	    ELSE (*Not External Control*)
	        IF Robot.Outputs.MotionControl.MoveID = 32120 THEN
	            Robot.Outputs.MotionControl.MoveID := 32121;
	        ELSIF Robot.Outputs.MotionControl.MoveID = 32121 THEN
	            Robot.Outputs.MotionControl.MoveID := 32120;
	        ELSIF Robot.Outputs.MotionControl.MoveID <> 32120 OR Robot.Outputs.MotionControl.MoveID <> 32121 THEN
	            Robot.Outputs.MotionControl.MoveID := 32120;
	        END_IF;
	        Sent := TRUE;
	    END_IF;
	END_IF;

	(* Check if command has been sent, if so, check if it was received *)
	IF Sent AND
	    Robot.Outputs.MotionCommand.MoveCommand = EnumToNum(Meca500Cmd#SetCartAcc) AND
	    Robot.Outputs.MotionCommand.MoveSubIndex001 = Output_Params[1] AND 
		Robot.Outputs.MotionCommand.MoveSubIndex002 = Output_Params[2] AND 
		Robot.Outputs.MotionCommand.MoveSubIndex003 = Output_Params[3] AND 
		Robot.Outputs.MotionCommand.MoveSubIndex004 = Output_Params[4] AND 
		Robot.Outputs.MotionCommand.MoveSubIndex005 = Output_Params[5] AND 
		Robot.Outputs.MotionCommand.MoveSubIndex006 = Output_Params[6] AND
		Robot.Inputs.Motion.MoveID = Robot.Outputs.MotionControl.MoveID 
	THEN
		 Buffered := TRUE;
	END_IF;


	(*If External _Move ID is equal to Internal, raise an error*)
	IF ExternalMoveID = 32120 OR ExternalMoveID = 32121 THEN
	    Error := TRUE;
	END_IF;

	FirstScan := TRUE;
ELSE
	FirstScan := False;
	Sent := FALSE;
	Buffered := FALSE;
END_IF;
END_FUNCTION_BLOCK

FUNCTION_BLOCK Meca500_SetCartAngVel
VAR
    Output_Params : array[1..6] of real;
    FirstScan : BOOL := False;
END_VAR
VAR_INPUT
    Execute : BOOL;
    Velocity_Limit : REAL;
END_VAR
VAR_OUTPUT
    Sent : BOOL;
    Buffered : BOOL;
    Error : BOOL;
END_VAR
VAR_IN_OUT
    Robot : Meca500;
END_VAR
VAR_INPUT
    ExternalStateControl : BOOL;
    ExternalMoveID : UINT;
END_VAR
IF Execute THEN	
	(*Collect Inputs and store them locally*)
	Output_Params[1]:=Velocity_Limit;
	Output_Params[2]:=0;
	Output_Params[3]:=0;
	Output_Params[4]:=0;
	Output_Params[5]:=0;
	Output_Params[6]:=0;

	(* If Values have change, Reinitialise Outputs*)

	IF FirstScan=0 OR 
		Robot.Outputs.MotionCommand.MoveSubIndex001 <> Output_Params[1] OR 
		Robot.Outputs.MotionCommand.MoveSubIndex002 <> Output_Params[2] OR 
		Robot.Outputs.MotionCommand.MoveSubIndex003 <> Output_Params[3] OR
		Robot.Outputs.MotionCommand.MoveSubIndex004 <> Output_Params[4] OR 
		Robot.Outputs.MotionCommand.MoveSubIndex005 <> Output_Params[5] OR 
		Robot.Outputs.MotionCommand.MoveSubIndex006 <> Output_Params[6] 
	THEN
		Buffered := FALSE;
		Sent := FALSE;
	END_IF;


	(*if not in legacy mode, Act Setpoint*)
	IF Robot.Outputs.MotionControl.MoveID <> 0 THEN
	    Robot.Outputs.MotionControl.SetPoint := TRUE;
	END_IF;

	(* To send _Move, send _Move ID *)
	IF NOT Buffered AND NOT Sent THEN
	    
	    Robot.Outputs.MotionCommand.MoveCommand	:= EnumToNum(Meca500Cmd#SetCartAngVel);
	    Robot.Outputs.MotionCommand.MoveSubIndex001 := Output_Params[1];
		Robot.Outputs.MotionCommand.MoveSubIndex002 := Output_Params[2];
		Robot.Outputs.MotionCommand.MoveSubIndex003 := Output_Params[3];
		Robot.Outputs.MotionCommand.MoveSubIndex004 := Output_Params[4];
		Robot.Outputs.MotionCommand.MoveSubIndex005 := Output_Params[5];
		Robot.Outputs.MotionCommand.MoveSubIndex006 := Output_Params[6];
	    
	    IF ExternalStateControl THEN
	        IF ExternalMoveID <> 0 AND ExternalMoveID <> 32100 AND ExternalMoveID <> 32101 THEN
	            Robot.Outputs.MotionControl.MoveID := ExternalMoveID;
	            Sent := TRUE;
	        END_IF;
	        
	    ELSE (*Not External Control*)
	        IF Robot.Outputs.MotionControl.MoveID = 32100 THEN
	            Robot.Outputs.MotionControl.MoveID := 32101;
	        ELSIF Robot.Outputs.MotionControl.MoveID = 32101 THEN
	            Robot.Outputs.MotionControl.MoveID := 32100;
	        ELSIF Robot.Outputs.MotionControl.MoveID <> 32100 OR Robot.Outputs.MotionControl.MoveID <> 32101 THEN
	            Robot.Outputs.MotionControl.MoveID := 32100;
	        END_IF;
	        Sent := TRUE;
	    END_IF;
	END_IF;

	(* Check if command has been sent, if so, check if it was received *)
	IF Sent AND
	    Robot.Outputs.MotionCommand.MoveCommand = EnumToNum(Meca500Cmd#SetCartAngVel) AND
	    Robot.Outputs.MotionCommand.MoveSubIndex001 = Output_Params[1] AND 
		Robot.Outputs.MotionCommand.MoveSubIndex002 = Output_Params[2] AND 
		Robot.Outputs.MotionCommand.MoveSubIndex003 = Output_Params[3] AND 
		Robot.Outputs.MotionCommand.MoveSubIndex004 = Output_Params[4] AND 
		Robot.Outputs.MotionCommand.MoveSubIndex005 = Output_Params[5] AND 
		Robot.Outputs.MotionCommand.MoveSubIndex006 = Output_Params[6] AND
		Robot.Inputs.Motion.MoveID = Robot.Outputs.MotionControl.MoveID 
	THEN
		 Buffered := TRUE;
	END_IF;


	(*If External _Move ID is equal to Internal, raise an error*)
	IF ExternalMoveID = 32100 OR ExternalMoveID = 32101 THEN
	    Error := TRUE;
	END_IF;

	FirstScan := TRUE;
ELSE
	FirstScan := False;
	Sent := FALSE;
	Buffered := FALSE;
END_IF;
END_FUNCTION_BLOCK

FUNCTION_BLOCK Meca500_SetCartLinVel
VAR
    Output_Params : array[1..6] of real;
    FirstScan : BOOL := False;
END_VAR
VAR_INPUT
    Execute : BOOL;
    Velocity_Limit : REAL;
END_VAR
VAR_OUTPUT
    Sent : BOOL;
    Buffered : BOOL;
    Error : BOOL;
END_VAR
VAR_IN_OUT
    Robot : Meca500;
END_VAR
VAR_INPUT
    ExternalStateControl : BOOL;
    ExternalMoveID : UINT;
END_VAR
IF Execute THEN	
	(*Collect Inputs and store them locally*)
	Output_Params[1]:=Velocity_Limit;
	Output_Params[2]:=0;
	Output_Params[3]:=0;
	Output_Params[4]:=0;
	Output_Params[5]:=0;
	Output_Params[6]:=0;

	(* If Values have change, Reinitialise Outputs*)

	IF FirstScan=0 OR 
		Robot.Outputs.MotionCommand.MoveSubIndex001 <> Output_Params[1] OR 
		Robot.Outputs.MotionCommand.MoveSubIndex002 <> Output_Params[2] OR 
		Robot.Outputs.MotionCommand.MoveSubIndex003 <> Output_Params[3] OR
		Robot.Outputs.MotionCommand.MoveSubIndex004 <> Output_Params[4] OR 
		Robot.Outputs.MotionCommand.MoveSubIndex005 <> Output_Params[5] OR 
		Robot.Outputs.MotionCommand.MoveSubIndex006 <> Output_Params[6] 
	THEN
		Buffered := FALSE;
		Sent := FALSE;
	END_IF;


	(*if not in legacy mode, Act Setpoint*)
	IF Robot.Outputs.MotionControl.MoveID <> 0 THEN
	    Robot.Outputs.MotionControl.SetPoint := TRUE;
	END_IF;

	(* To send _Move, send _Move ID *)
	IF NOT Buffered AND NOT Sent THEN
	    
	    Robot.Outputs.MotionCommand.MoveCommand	:= EnumToNum(Meca500Cmd#SetCartLinVel);
	    Robot.Outputs.MotionCommand.MoveSubIndex001 := Output_Params[1];
		Robot.Outputs.MotionCommand.MoveSubIndex002 := Output_Params[2];
		Robot.Outputs.MotionCommand.MoveSubIndex003 := Output_Params[3];
		Robot.Outputs.MotionCommand.MoveSubIndex004 := Output_Params[4];
		Robot.Outputs.MotionCommand.MoveSubIndex005 := Output_Params[5];
		Robot.Outputs.MotionCommand.MoveSubIndex006 := Output_Params[6];
	    
	    IF ExternalStateControl THEN
	        IF ExternalMoveID <> 0 AND ExternalMoveID <> 32110 AND ExternalMoveID <> 32111 THEN
	            Robot.Outputs.MotionControl.MoveID := ExternalMoveID;
	            Sent := TRUE;
	        END_IF;
	        
	    ELSE (*Not External Control*)
	        IF Robot.Outputs.MotionControl.MoveID = 32110 THEN
	            Robot.Outputs.MotionControl.MoveID := 32111;
	        ELSIF Robot.Outputs.MotionControl.MoveID = 32111 THEN
	            Robot.Outputs.MotionControl.MoveID := 32110;
	        ELSIF Robot.Outputs.MotionControl.MoveID <> 32110 OR Robot.Outputs.MotionControl.MoveID <> 32111 THEN
	            Robot.Outputs.MotionControl.MoveID := 32110;
	        END_IF;
	        Sent := TRUE;
	    END_IF;
	END_IF;

	(* Check if command has been sent, if so, check if it was received *)
	IF Sent AND
	    Robot.Outputs.MotionCommand.MoveCommand = EnumToNum(Meca500Cmd#SetCartLinVel) AND
	    Robot.Outputs.MotionCommand.MoveSubIndex001 = Output_Params[1] AND 
		Robot.Outputs.MotionCommand.MoveSubIndex002 = Output_Params[2] AND 
		Robot.Outputs.MotionCommand.MoveSubIndex003 = Output_Params[3] AND 
		Robot.Outputs.MotionCommand.MoveSubIndex004 = Output_Params[4] AND 
		Robot.Outputs.MotionCommand.MoveSubIndex005 = Output_Params[5] AND 
		Robot.Outputs.MotionCommand.MoveSubIndex006 = Output_Params[6] AND
		Robot.Inputs.Motion.MoveID = Robot.Outputs.MotionControl.MoveID 
	THEN
		 Buffered := TRUE;
	END_IF;


	(*If External _Move ID is equal to Internal, raise an error*)
	IF ExternalMoveID = 32110 OR ExternalMoveID = 32111 THEN
	    Error := TRUE;
	END_IF;

	FirstScan := TRUE;
ELSE
	FirstScan := False;
	Sent := FALSE;
	Buffered := FALSE;
END_IF;
END_FUNCTION_BLOCK

FUNCTION_BLOCK Meca500_SetCheckpoint
VAR
    Output_Params : array[1..6] of real;
    FirstScan : BOOL := False;
END_VAR
VAR_INPUT
    Execute : BOOL;
    CheckpointID : REAL;
END_VAR
VAR_OUTPUT
    Sent : BOOL;
    Buffered : BOOL;
    Error : BOOL;
END_VAR
VAR_IN_OUT
    Robot : Meca500;
END_VAR
VAR_INPUT
    ExternalStateControl : BOOL;
    ExternalMoveID : UINT;
END_VAR
IF Execute THEN	
	(*Collect Inputs and store them locally*)
	Output_Params[1]:=CheckpointID;
	Output_Params[2]:=0;
	Output_Params[3]:=0;
	Output_Params[4]:=0;
	Output_Params[5]:=0;
	Output_Params[6]:=0;

	(* If Values have change, Reinitialise Outputs*)

	IF FirstScan=0 OR 
		Robot.Outputs.MotionCommand.MoveSubIndex001 <> Output_Params[1] OR 
		Robot.Outputs.MotionCommand.MoveSubIndex002 <> Output_Params[2] OR 
		Robot.Outputs.MotionCommand.MoveSubIndex003 <> Output_Params[3] OR
		Robot.Outputs.MotionCommand.MoveSubIndex004 <> Output_Params[4] OR 
		Robot.Outputs.MotionCommand.MoveSubIndex005 <> Output_Params[5] OR 
		Robot.Outputs.MotionCommand.MoveSubIndex006 <> Output_Params[6] 
	THEN
		Buffered := FALSE;
		Sent := FALSE;
	END_IF;


	(*if not in legacy mode, Act Setpoint*)
	IF Robot.Outputs.MotionControl.MoveID <> 0 THEN
	    Robot.Outputs.MotionControl.SetPoint := TRUE;
	END_IF;

	(* To send _Move, send _Move ID *)
	IF NOT Buffered AND NOT Sent THEN
	    
	    Robot.Outputs.MotionCommand.MoveCommand	:= EnumToNum(Meca500Cmd#SetCheckpoint);
	    Robot.Outputs.MotionCommand.MoveSubIndex001 := Output_Params[1];
		Robot.Outputs.MotionCommand.MoveSubIndex002 := Output_Params[2];
		Robot.Outputs.MotionCommand.MoveSubIndex003 := Output_Params[3];
		Robot.Outputs.MotionCommand.MoveSubIndex004 := Output_Params[4];
		Robot.Outputs.MotionCommand.MoveSubIndex005 := Output_Params[5];
		Robot.Outputs.MotionCommand.MoveSubIndex006 := Output_Params[6];
	    
	    IF ExternalStateControl THEN
	        IF ExternalMoveID <> 0 AND ExternalMoveID <> 32170 AND ExternalMoveID <> 32171 THEN
	            Robot.Outputs.MotionControl.MoveID := ExternalMoveID;
	            Sent := TRUE;
	        END_IF;
	        
	    ELSE (*Not External Control*)
	        IF Robot.Outputs.MotionControl.MoveID = 32170 THEN
	            Robot.Outputs.MotionControl.MoveID := 32171;
	        ELSIF Robot.Outputs.MotionControl.MoveID = 32171 THEN
	            Robot.Outputs.MotionControl.MoveID := 32170;
	        ELSIF Robot.Outputs.MotionControl.MoveID <> 32170 OR Robot.Outputs.MotionControl.MoveID <> 32171 THEN
	            Robot.Outputs.MotionControl.MoveID := 32170;
	        END_IF;
	        Sent := TRUE;
	    END_IF;
	END_IF;

	(* Check if command has been sent, if so, check if it was received *)
	IF Sent AND
	    Robot.Outputs.MotionCommand.MoveCommand = EnumToNum(Meca500Cmd#SetCheckpoint) AND
	    Robot.Outputs.MotionCommand.MoveSubIndex001 = Output_Params[1] AND 
		Robot.Outputs.MotionCommand.MoveSubIndex002 = Output_Params[2] AND 
		Robot.Outputs.MotionCommand.MoveSubIndex003 = Output_Params[3] AND 
		Robot.Outputs.MotionCommand.MoveSubIndex004 = Output_Params[4] AND 
		Robot.Outputs.MotionCommand.MoveSubIndex005 = Output_Params[5] AND 
		Robot.Outputs.MotionCommand.MoveSubIndex006 = Output_Params[6] AND
		Robot.Inputs.Motion.MoveID = Robot.Outputs.MotionControl.MoveID 
	THEN
		 Buffered := TRUE;
	END_IF;


	(*If External _Move ID is equal to Internal, raise an error*)
	IF ExternalMoveID = 32170 OR ExternalMoveID = 32171 THEN
	    Error := TRUE;
	END_IF;

	FirstScan := TRUE;
ELSE
	FirstScan := False;
	Sent := FALSE;
	Buffered := FALSE;
END_IF;
END_FUNCTION_BLOCK

FUNCTION_BLOCK Meca500_SetConf
VAR
    Output_Params : array[1..6] of real;
    FirstScan : BOOL := False;
END_VAR
VAR_INPUT
    Execute : BOOL;
    Shoulder : REAL;
    Elbow : REAL;
    Wrist : REAL;
END_VAR
VAR_OUTPUT
    Sent : BOOL;
    Buffered : BOOL;
    Error : BOOL;
END_VAR
VAR_IN_OUT
    Robot : Meca500;
END_VAR
VAR_INPUT
    ExternalStateControl : BOOL;
    ExternalMoveID : UINT;
END_VAR
IF Execute THEN	
	(*Collect Inputs and store them locally*)
	Output_Params[1]:=Shoulder;
	Output_Params[2]:=Elbow;
	Output_Params[3]:=Wrist;
	Output_Params[4]:=0;
	Output_Params[5]:=0;
	Output_Params[6]:=0;

	(* If Values have change, Reinitialise Outputs*)

	IF FirstScan=0 OR 
		Robot.Outputs.MotionCommand.MoveSubIndex001 <> Output_Params[1] OR 
		Robot.Outputs.MotionCommand.MoveSubIndex002 <> Output_Params[2] OR 
		Robot.Outputs.MotionCommand.MoveSubIndex003 <> Output_Params[3] OR
		Robot.Outputs.MotionCommand.MoveSubIndex004 <> Output_Params[4] OR 
		Robot.Outputs.MotionCommand.MoveSubIndex005 <> Output_Params[5] OR 
		Robot.Outputs.MotionCommand.MoveSubIndex006 <> Output_Params[6] 
	THEN
		Buffered := FALSE;
		Sent := FALSE;
	END_IF;


	(*if not in legacy mode, Act Setpoint*)
	IF Robot.Outputs.MotionControl.MoveID <> 0 THEN
	    Robot.Outputs.MotionControl.SetPoint := TRUE;
	END_IF;

	(* To send _Move, send _Move ID *)
	IF NOT Buffered AND NOT Sent THEN
	    
	    Robot.Outputs.MotionCommand.MoveCommand	:= EnumToNum(Meca500Cmd#SetConf);
	    Robot.Outputs.MotionCommand.MoveSubIndex001 := Output_Params[1];
		Robot.Outputs.MotionCommand.MoveSubIndex002 := Output_Params[2];
		Robot.Outputs.MotionCommand.MoveSubIndex003 := Output_Params[3];
		Robot.Outputs.MotionCommand.MoveSubIndex004 := Output_Params[4];
		Robot.Outputs.MotionCommand.MoveSubIndex005 := Output_Params[5];
		Robot.Outputs.MotionCommand.MoveSubIndex006 := Output_Params[6];
	    
	    IF ExternalStateControl THEN
	        IF ExternalMoveID <> 0 AND ExternalMoveID <> 32150 AND ExternalMoveID <> 32151 THEN
	            Robot.Outputs.MotionControl.MoveID := ExternalMoveID;
	            Sent := TRUE;
	        END_IF;
	        
	    ELSE (*Not External Control*)
	        IF Robot.Outputs.MotionControl.MoveID = 32150 THEN
	            Robot.Outputs.MotionControl.MoveID := 32151;
	        ELSIF Robot.Outputs.MotionControl.MoveID = 32151 THEN
	            Robot.Outputs.MotionControl.MoveID := 32150;
	        ELSIF Robot.Outputs.MotionControl.MoveID <> 32150 OR Robot.Outputs.MotionControl.MoveID <> 32151 THEN
	            Robot.Outputs.MotionControl.MoveID := 32150;
	        END_IF;
	        Sent := TRUE;
	    END_IF;
	END_IF;

	(* Check if command has been sent, if so, check if it was received *)
	IF Sent AND
	    Robot.Outputs.MotionCommand.MoveCommand = EnumToNum(Meca500Cmd#SetConf) AND
	    Robot.Outputs.MotionCommand.MoveSubIndex001 = Output_Params[1] AND 
		Robot.Outputs.MotionCommand.MoveSubIndex002 = Output_Params[2] AND 
		Robot.Outputs.MotionCommand.MoveSubIndex003 = Output_Params[3] AND 
		Robot.Outputs.MotionCommand.MoveSubIndex004 = Output_Params[4] AND 
		Robot.Outputs.MotionCommand.MoveSubIndex005 = Output_Params[5] AND 
		Robot.Outputs.MotionCommand.MoveSubIndex006 = Output_Params[6] AND
		Robot.Inputs.Motion.MoveID = Robot.Outputs.MotionControl.MoveID 
	THEN
		 Buffered := TRUE;
	END_IF;


	(*If External _Move ID is equal to Internal, raise an error*)
	IF ExternalMoveID = 32150 OR ExternalMoveID = 32151 THEN
	    Error := TRUE;
	END_IF;

	FirstScan := TRUE;
ELSE
	FirstScan := False;
	Sent := FALSE;
	Buffered := FALSE;
END_IF;
END_FUNCTION_BLOCK

FUNCTION_BLOCK Meca500_SetConfTurn
VAR
    Output_Params : array[1..6] of real;
    FirstScan : BOOL := False;
END_VAR
VAR_INPUT
    Execute : BOOL;
    Config : REAL;
END_VAR
VAR_OUTPUT
    Sent : BOOL;
    Buffered : BOOL;
    Error : BOOL;
END_VAR
VAR_IN_OUT
    Robot : Meca500;
END_VAR
VAR_INPUT
    ExternalStateControl : BOOL;
    ExternalMoveID : UINT;
END_VAR
IF Execute THEN	
	(*Collect Inputs and store them locally*)
	Output_Params[1]:=Config;
	Output_Params[2]:=0;
	Output_Params[3]:=0;
	Output_Params[4]:=0;
	Output_Params[5]:=0;
	Output_Params[6]:=0;

	(* If Values have change, Reinitialise Outputs*)

	IF FirstScan=0 OR 
		Robot.Outputs.MotionCommand.MoveSubIndex001 <> Output_Params[1] OR 
		Robot.Outputs.MotionCommand.MoveSubIndex002 <> Output_Params[2] OR 
		Robot.Outputs.MotionCommand.MoveSubIndex003 <> Output_Params[3] OR
		Robot.Outputs.MotionCommand.MoveSubIndex004 <> Output_Params[4] OR 
		Robot.Outputs.MotionCommand.MoveSubIndex005 <> Output_Params[5] OR 
		Robot.Outputs.MotionCommand.MoveSubIndex006 <> Output_Params[6] 
	THEN
		Buffered := FALSE;
		Sent := FALSE;
	END_IF;


	(*if not in legacy mode, Act Setpoint*)
	IF Robot.Outputs.MotionControl.MoveID <> 0 THEN
	    Robot.Outputs.MotionControl.SetPoint := TRUE;
	END_IF;

	(* To send _Move, send _Move ID *)
	IF NOT Buffered AND NOT Sent THEN
	    
	    Robot.Outputs.MotionCommand.MoveCommand	:= EnumToNum(Meca500Cmd#SetConfTurn);
	    Robot.Outputs.MotionCommand.MoveSubIndex001 := Output_Params[1];
		Robot.Outputs.MotionCommand.MoveSubIndex002 := Output_Params[2];
		Robot.Outputs.MotionCommand.MoveSubIndex003 := Output_Params[3];
		Robot.Outputs.MotionCommand.MoveSubIndex004 := Output_Params[4];
		Robot.Outputs.MotionCommand.MoveSubIndex005 := Output_Params[5];
		Robot.Outputs.MotionCommand.MoveSubIndex006 := Output_Params[6];
	    
	    IF ExternalStateControl THEN
	        IF ExternalMoveID <> 0 AND ExternalMoveID <> 32250 AND ExternalMoveID <> 32251 THEN
	            Robot.Outputs.MotionControl.MoveID := ExternalMoveID;
	            Sent := TRUE;
	        END_IF;
	        
	    ELSE (*Not External Control*)
	        IF Robot.Outputs.MotionControl.MoveID = 32250 THEN
	            Robot.Outputs.MotionControl.MoveID := 32251;
	        ELSIF Robot.Outputs.MotionControl.MoveID = 32251 THEN
	            Robot.Outputs.MotionControl.MoveID := 32250;
	        ELSIF Robot.Outputs.MotionControl.MoveID <> 32250 OR Robot.Outputs.MotionControl.MoveID <> 32251 THEN
	            Robot.Outputs.MotionControl.MoveID := 32250;
	        END_IF;
	        Sent := TRUE;
	    END_IF;
	END_IF;

	(* Check if command has been sent, if so, check if it was received *)
	IF Sent AND
	    Robot.Outputs.MotionCommand.MoveCommand = EnumToNum(Meca500Cmd#SetConfTurn) AND
	    Robot.Outputs.MotionCommand.MoveSubIndex001 = Output_Params[1] AND 
		Robot.Outputs.MotionCommand.MoveSubIndex002 = Output_Params[2] AND 
		Robot.Outputs.MotionCommand.MoveSubIndex003 = Output_Params[3] AND 
		Robot.Outputs.MotionCommand.MoveSubIndex004 = Output_Params[4] AND 
		Robot.Outputs.MotionCommand.MoveSubIndex005 = Output_Params[5] AND 
		Robot.Outputs.MotionCommand.MoveSubIndex006 = Output_Params[6] AND
		Robot.Inputs.Motion.MoveID = Robot.Outputs.MotionControl.MoveID 
	THEN
		 Buffered := TRUE;
	END_IF;


	(*If External _Move ID is equal to Internal, raise an error*)
	IF ExternalMoveID = 32250 OR ExternalMoveID = 32251 THEN
	    Error := TRUE;
	END_IF;

	FirstScan := TRUE;
ELSE
	FirstScan := False;
	Sent := FALSE;
	Buffered := FALSE;
END_IF;
END_FUNCTION_BLOCK

FUNCTION_BLOCK Meca500_SetGripperForce
VAR
    Output_Params : array[1..6] of real;
    FirstScan : BOOL := False;
END_VAR
VAR_INPUT
    Execute : BOOL;
    Force : REAL;
END_VAR
VAR_OUTPUT
    Sent : BOOL;
    Buffered : BOOL;
    Error : BOOL;
END_VAR
VAR_IN_OUT
    Robot : Meca500;
END_VAR
VAR_INPUT
    ExternalStateControl : BOOL;
    ExternalMoveID : UINT;
END_VAR
IF Execute THEN	
	(*Collect Inputs and store them locally*)
	Output_Params[1]:=Force;
	Output_Params[2]:=0;
	Output_Params[3]:=0;
	Output_Params[4]:=0;
	Output_Params[5]:=0;
	Output_Params[6]:=0;

	(* If Values have change, Reinitialise Outputs*)

	IF FirstScan=0 OR 
		Robot.Outputs.MotionCommand.MoveSubIndex001 <> Output_Params[1] OR 
		Robot.Outputs.MotionCommand.MoveSubIndex002 <> Output_Params[2] OR 
		Robot.Outputs.MotionCommand.MoveSubIndex003 <> Output_Params[3] OR
		Robot.Outputs.MotionCommand.MoveSubIndex004 <> Output_Params[4] OR 
		Robot.Outputs.MotionCommand.MoveSubIndex005 <> Output_Params[5] OR 
		Robot.Outputs.MotionCommand.MoveSubIndex006 <> Output_Params[6] 
	THEN
		Buffered := FALSE;
		Sent := FALSE;
	END_IF;


	(*if not in legacy mode, Act Setpoint*)
	IF Robot.Outputs.MotionControl.MoveID <> 0 THEN
	    Robot.Outputs.MotionControl.SetPoint := TRUE;
	END_IF;

	(* To send _Move, send _Move ID *)
	IF NOT Buffered AND NOT Sent THEN
	    
	    Robot.Outputs.MotionCommand.MoveCommand	:= EnumToNum(Meca500Cmd#SetGripperForce);
	    Robot.Outputs.MotionCommand.MoveSubIndex001 := Output_Params[1];
		Robot.Outputs.MotionCommand.MoveSubIndex002 := Output_Params[2];
		Robot.Outputs.MotionCommand.MoveSubIndex003 := Output_Params[3];
		Robot.Outputs.MotionCommand.MoveSubIndex004 := Output_Params[4];
		Robot.Outputs.MotionCommand.MoveSubIndex005 := Output_Params[5];
		Robot.Outputs.MotionCommand.MoveSubIndex006 := Output_Params[6];
	    
	    IF ExternalStateControl THEN
	        IF ExternalMoveID <> 0 AND ExternalMoveID <> 32200 AND ExternalMoveID <> 32201 THEN
	            Robot.Outputs.MotionControl.MoveID := ExternalMoveID;
	            Sent := TRUE;
	        END_IF;
	        
	    ELSE (*Not External Control*)
	        IF Robot.Outputs.MotionControl.MoveID = 32200 THEN
	            Robot.Outputs.MotionControl.MoveID := 32201;
	        ELSIF Robot.Outputs.MotionControl.MoveID = 32201 THEN
	            Robot.Outputs.MotionControl.MoveID := 32200;
	        ELSIF Robot.Outputs.MotionControl.MoveID <> 32200 OR Robot.Outputs.MotionControl.MoveID <> 32201 THEN
	            Robot.Outputs.MotionControl.MoveID := 32200;
	        END_IF;
	        Sent := TRUE;
	    END_IF;
	END_IF;

	(* Check if command has been sent, if so, check if it was received *)
	IF Sent AND
	    Robot.Outputs.MotionCommand.MoveCommand = EnumToNum(Meca500Cmd#SetGripperForce) AND
	    Robot.Outputs.MotionCommand.MoveSubIndex001 = Output_Params[1] AND 
		Robot.Outputs.MotionCommand.MoveSubIndex002 = Output_Params[2] AND 
		Robot.Outputs.MotionCommand.MoveSubIndex003 = Output_Params[3] AND 
		Robot.Outputs.MotionCommand.MoveSubIndex004 = Output_Params[4] AND 
		Robot.Outputs.MotionCommand.MoveSubIndex005 = Output_Params[5] AND 
		Robot.Outputs.MotionCommand.MoveSubIndex006 = Output_Params[6] AND
		Robot.Inputs.Motion.MoveID = Robot.Outputs.MotionControl.MoveID 
	THEN
		 Buffered := TRUE;
	END_IF;


	(*If External _Move ID is equal to Internal, raise an error*)
	IF ExternalMoveID = 32200 OR ExternalMoveID = 32201 THEN
	    Error := TRUE;
	END_IF;

	FirstScan := TRUE;
ELSE
	FirstScan := False;
	Sent := FALSE;
	Buffered := FALSE;
END_IF;
END_FUNCTION_BLOCK

FUNCTION_BLOCK Meca500_SetGripperRange
VAR
    Output_Params : array[1..6] of real;
    FirstScan : BOOL := False;
END_VAR
VAR_INPUT
    Execute : BOOL;
    Minimum : REAL;
    Maximum : REAL;
END_VAR
VAR_OUTPUT
    Sent : BOOL;
    Buffered : BOOL;
    Error : BOOL;
END_VAR
VAR_IN_OUT
    Robot : Meca500;
END_VAR
VAR_INPUT
    ExternalStateControl : BOOL;
    ExternalMoveID : UINT;
END_VAR
IF Execute THEN	
	(*Collect Inputs and store them locally*)
	Output_Params[1]:=Minimum;
	Output_Params[2]:=Maximum;
	Output_Params[3]:=0;
	Output_Params[4]:=0;
	Output_Params[5]:=0;
	Output_Params[6]:=0;

	(* If Values have change, Reinitialise Outputs*)

	IF FirstScan=0 OR 
		Robot.Outputs.MotionCommand.MoveSubIndex001 <> Output_Params[1] OR 
		Robot.Outputs.MotionCommand.MoveSubIndex002 <> Output_Params[2] OR 
		Robot.Outputs.MotionCommand.MoveSubIndex003 <> Output_Params[3] OR
		Robot.Outputs.MotionCommand.MoveSubIndex004 <> Output_Params[4] OR 
		Robot.Outputs.MotionCommand.MoveSubIndex005 <> Output_Params[5] OR 
		Robot.Outputs.MotionCommand.MoveSubIndex006 <> Output_Params[6] 
	THEN
		Buffered := FALSE;
		Sent := FALSE;
	END_IF;


	(*if not in legacy mode, Act Setpoint*)
	IF Robot.Outputs.MotionControl.MoveID <> 0 THEN
	    Robot.Outputs.MotionControl.SetPoint := TRUE;
	END_IF;

	(* To send _Move, send _Move ID *)
	IF NOT Buffered AND NOT Sent THEN
	    
	    Robot.Outputs.MotionCommand.MoveCommand	:= EnumToNum(Meca500Cmd#SetGripperRange);
	    Robot.Outputs.MotionCommand.MoveSubIndex001 := Output_Params[1];
		Robot.Outputs.MotionCommand.MoveSubIndex002 := Output_Params[2];
		Robot.Outputs.MotionCommand.MoveSubIndex003 := Output_Params[3];
		Robot.Outputs.MotionCommand.MoveSubIndex004 := Output_Params[4];
		Robot.Outputs.MotionCommand.MoveSubIndex005 := Output_Params[5];
		Robot.Outputs.MotionCommand.MoveSubIndex006 := Output_Params[6];
	    
	    IF ExternalStateControl THEN
	        IF ExternalMoveID <> 0 AND ExternalMoveID <> 32310 AND ExternalMoveID <> 32311 THEN
	            Robot.Outputs.MotionControl.MoveID := ExternalMoveID;
	            Sent := TRUE;
	        END_IF;
	        
	    ELSE (*Not External Control*)
	        IF Robot.Outputs.MotionControl.MoveID = 32310 THEN
	            Robot.Outputs.MotionControl.MoveID := 32311;
	        ELSIF Robot.Outputs.MotionControl.MoveID = 32311 THEN
	            Robot.Outputs.MotionControl.MoveID := 32310;
	        ELSIF Robot.Outputs.MotionControl.MoveID <> 32310 OR Robot.Outputs.MotionControl.MoveID <> 32311 THEN
	            Robot.Outputs.MotionControl.MoveID := 32310;
	        END_IF;
	        Sent := TRUE;
	    END_IF;
	END_IF;

	(* Check if command has been sent, if so, check if it was received *)
	IF Sent AND
	    Robot.Outputs.MotionCommand.MoveCommand = EnumToNum(Meca500Cmd#SetGripperRange) AND
	    Robot.Outputs.MotionCommand.MoveSubIndex001 = Output_Params[1] AND 
		Robot.Outputs.MotionCommand.MoveSubIndex002 = Output_Params[2] AND 
		Robot.Outputs.MotionCommand.MoveSubIndex003 = Output_Params[3] AND 
		Robot.Outputs.MotionCommand.MoveSubIndex004 = Output_Params[4] AND 
		Robot.Outputs.MotionCommand.MoveSubIndex005 = Output_Params[5] AND 
		Robot.Outputs.MotionCommand.MoveSubIndex006 = Output_Params[6] AND
		Robot.Inputs.Motion.MoveID = Robot.Outputs.MotionControl.MoveID 
	THEN
		 Buffered := TRUE;
	END_IF;


	(*If External _Move ID is equal to Internal, raise an error*)
	IF ExternalMoveID = 32310 OR ExternalMoveID = 32311 THEN
	    Error := TRUE;
	END_IF;

	FirstScan := TRUE;
ELSE
	FirstScan := False;
	Sent := FALSE;
	Buffered := FALSE;
END_IF;
END_FUNCTION_BLOCK

FUNCTION_BLOCK Meca500_SetGripperVel
VAR
    Output_Params : array[1..6] of real;
    FirstScan : BOOL := False;
END_VAR
VAR_INPUT
    Execute : BOOL;
    Speed : REAL;
END_VAR
VAR_OUTPUT
    Sent : BOOL;
    Buffered : BOOL;
    Error : BOOL;
END_VAR
VAR_IN_OUT
    Robot : Meca500;
END_VAR
VAR_INPUT
    ExternalStateControl : BOOL;
    ExternalMoveID : UINT;
END_VAR
IF Execute THEN	
	(*Collect Inputs and store them locally*)
	Output_Params[1]:=Speed;
	Output_Params[2]:=0;
	Output_Params[3]:=0;
	Output_Params[4]:=0;
	Output_Params[5]:=0;
	Output_Params[6]:=0;

	(* If Values have change, Reinitialise Outputs*)

	IF FirstScan=0 OR 
		Robot.Outputs.MotionCommand.MoveSubIndex001 <> Output_Params[1] OR 
		Robot.Outputs.MotionCommand.MoveSubIndex002 <> Output_Params[2] OR 
		Robot.Outputs.MotionCommand.MoveSubIndex003 <> Output_Params[3] OR
		Robot.Outputs.MotionCommand.MoveSubIndex004 <> Output_Params[4] OR 
		Robot.Outputs.MotionCommand.MoveSubIndex005 <> Output_Params[5] OR 
		Robot.Outputs.MotionCommand.MoveSubIndex006 <> Output_Params[6] 
	THEN
		Buffered := FALSE;
		Sent := FALSE;
	END_IF;


	(*if not in legacy mode, Act Setpoint*)
	IF Robot.Outputs.MotionControl.MoveID <> 0 THEN
	    Robot.Outputs.MotionControl.SetPoint := TRUE;
	END_IF;

	(* To send _Move, send _Move ID *)
	IF NOT Buffered AND NOT Sent THEN
	    
	    Robot.Outputs.MotionCommand.MoveCommand	:= EnumToNum(Meca500Cmd#SetGripperVel);
	    Robot.Outputs.MotionCommand.MoveSubIndex001 := Output_Params[1];
		Robot.Outputs.MotionCommand.MoveSubIndex002 := Output_Params[2];
		Robot.Outputs.MotionCommand.MoveSubIndex003 := Output_Params[3];
		Robot.Outputs.MotionCommand.MoveSubIndex004 := Output_Params[4];
		Robot.Outputs.MotionCommand.MoveSubIndex005 := Output_Params[5];
		Robot.Outputs.MotionCommand.MoveSubIndex006 := Output_Params[6];
	    
	    IF ExternalStateControl THEN
	        IF ExternalMoveID <> 0 AND ExternalMoveID <> 32190 AND ExternalMoveID <> 32191 THEN
	            Robot.Outputs.MotionControl.MoveID := ExternalMoveID;
	            Sent := TRUE;
	        END_IF;
	        
	    ELSE (*Not External Control*)
	        IF Robot.Outputs.MotionControl.MoveID = 32190 THEN
	            Robot.Outputs.MotionControl.MoveID := 32191;
	        ELSIF Robot.Outputs.MotionControl.MoveID = 32191 THEN
	            Robot.Outputs.MotionControl.MoveID := 32190;
	        ELSIF Robot.Outputs.MotionControl.MoveID <> 32190 OR Robot.Outputs.MotionControl.MoveID <> 32191 THEN
	            Robot.Outputs.MotionControl.MoveID := 32190;
	        END_IF;
	        Sent := TRUE;
	    END_IF;
	END_IF;

	(* Check if command has been sent, if so, check if it was received *)
	IF Sent AND
	    Robot.Outputs.MotionCommand.MoveCommand = EnumToNum(Meca500Cmd#SetGripperVel) AND
	    Robot.Outputs.MotionCommand.MoveSubIndex001 = Output_Params[1] AND 
		Robot.Outputs.MotionCommand.MoveSubIndex002 = Output_Params[2] AND 
		Robot.Outputs.MotionCommand.MoveSubIndex003 = Output_Params[3] AND 
		Robot.Outputs.MotionCommand.MoveSubIndex004 = Output_Params[4] AND 
		Robot.Outputs.MotionCommand.MoveSubIndex005 = Output_Params[5] AND 
		Robot.Outputs.MotionCommand.MoveSubIndex006 = Output_Params[6] AND
		Robot.Inputs.Motion.MoveID = Robot.Outputs.MotionControl.MoveID 
	THEN
		 Buffered := TRUE;
	END_IF;


	(*If External _Move ID is equal to Internal, raise an error*)
	IF ExternalMoveID = 32190 OR ExternalMoveID = 32191 THEN
	    Error := TRUE;
	END_IF;

	FirstScan := TRUE;
ELSE
	FirstScan := False;
	Sent := FALSE;
	Buffered := FALSE;
END_IF;
END_FUNCTION_BLOCK

FUNCTION_BLOCK Meca500_SetJointsAcc
VAR
    Output_Params : array[1..6] of real;
    FirstScan : BOOL := False;
END_VAR
VAR_INPUT
    Execute : BOOL;
    Acceleration_Percentage : REAL;
END_VAR
VAR_OUTPUT
    Sent : BOOL;
    Buffered : BOOL;
    Error : BOOL;
END_VAR
VAR_IN_OUT
    Robot : Meca500;
END_VAR
VAR_INPUT
    ExternalStateControl : BOOL;
    ExternalMoveID : UINT;
END_VAR
IF Execute THEN	
	(*Collect Inputs and store them locally*)
	Output_Params[1]:=Acceleration_Percentage;
	Output_Params[2]:=0;
	Output_Params[3]:=0;
	Output_Params[4]:=0;
	Output_Params[5]:=0;
	Output_Params[6]:=0;

	(* If Values have change, Reinitialise Outputs*)

	IF FirstScan=0 OR 
		Robot.Outputs.MotionCommand.MoveSubIndex001 <> Output_Params[1] OR 
		Robot.Outputs.MotionCommand.MoveSubIndex002 <> Output_Params[2] OR 
		Robot.Outputs.MotionCommand.MoveSubIndex003 <> Output_Params[3] OR
		Robot.Outputs.MotionCommand.MoveSubIndex004 <> Output_Params[4] OR 
		Robot.Outputs.MotionCommand.MoveSubIndex005 <> Output_Params[5] OR 
		Robot.Outputs.MotionCommand.MoveSubIndex006 <> Output_Params[6] 
	THEN
		Buffered := FALSE;
		Sent := FALSE;
	END_IF;


	(*if not in legacy mode, Act Setpoint*)
	IF Robot.Outputs.MotionControl.MoveID <> 0 THEN
	    Robot.Outputs.MotionControl.SetPoint := TRUE;
	END_IF;

	(* To send _Move, send _Move ID *)
	IF NOT Buffered AND NOT Sent THEN
	    
	    Robot.Outputs.MotionCommand.MoveCommand	:= EnumToNum(Meca500Cmd#SetJointAcc);
	    Robot.Outputs.MotionCommand.MoveSubIndex001 := Output_Params[1];
		Robot.Outputs.MotionCommand.MoveSubIndex002 := Output_Params[2];
		Robot.Outputs.MotionCommand.MoveSubIndex003 := Output_Params[3];
		Robot.Outputs.MotionCommand.MoveSubIndex004 := Output_Params[4];
		Robot.Outputs.MotionCommand.MoveSubIndex005 := Output_Params[5];
		Robot.Outputs.MotionCommand.MoveSubIndex006 := Output_Params[6];
	    
	    IF ExternalStateControl THEN
	        IF ExternalMoveID <> 0 AND ExternalMoveID <> 32090 AND ExternalMoveID <> 32091 THEN
	            Robot.Outputs.MotionControl.MoveID := ExternalMoveID;
	            Sent := TRUE;
	        END_IF;
	        
	    ELSE (*Not External Control*)
	        IF Robot.Outputs.MotionControl.MoveID = 32090 THEN
	            Robot.Outputs.MotionControl.MoveID := 32091;
	        ELSIF Robot.Outputs.MotionControl.MoveID = 32091 THEN
	            Robot.Outputs.MotionControl.MoveID := 32090;
	        ELSIF Robot.Outputs.MotionControl.MoveID <> 32090 OR Robot.Outputs.MotionControl.MoveID <> 32091 THEN
	            Robot.Outputs.MotionControl.MoveID := 32090;
	        END_IF;
	        Sent := TRUE;
	    END_IF;
	END_IF;

	(* Check if command has been sent, if so, check if it was received *)
	IF Sent AND
	    Robot.Outputs.MotionCommand.MoveCommand = EnumToNum(Meca500Cmd#SetJointAcc) AND
	    Robot.Outputs.MotionCommand.MoveSubIndex001 = Output_Params[1] AND 
		Robot.Outputs.MotionCommand.MoveSubIndex002 = Output_Params[2] AND 
		Robot.Outputs.MotionCommand.MoveSubIndex003 = Output_Params[3] AND 
		Robot.Outputs.MotionCommand.MoveSubIndex004 = Output_Params[4] AND 
		Robot.Outputs.MotionCommand.MoveSubIndex005 = Output_Params[5] AND 
		Robot.Outputs.MotionCommand.MoveSubIndex006 = Output_Params[6] AND
		Robot.Inputs.Motion.MoveID = Robot.Outputs.MotionControl.MoveID 
	THEN
		 Buffered := TRUE;
	END_IF;


	(*If External _Move ID is equal to Internal, raise an error*)
	IF ExternalMoveID = 32090 OR ExternalMoveID = 32091 THEN
	    Error := TRUE;
	END_IF;

	FirstScan := TRUE;
ELSE
	FirstScan := False;
	Sent := FALSE;
	Buffered := FALSE;
END_IF;
END_FUNCTION_BLOCK

FUNCTION_BLOCK Meca500_SetJointsVel
VAR
    Output_Params : array[1..6] of real;
    FirstScan : BOOL := False;
END_VAR
VAR_INPUT
    Execute : BOOL;
    Velocity_Percentage : REAL;
END_VAR
VAR_OUTPUT
    Sent : BOOL;
    Buffered : BOOL;
    Error : BOOL;
END_VAR
VAR_IN_OUT
    Robot : Meca500;
END_VAR
VAR_INPUT
    ExternalStateControl : BOOL;
    ExternalMoveID : UINT;
END_VAR
IF Execute THEN	
	(*Collect Inputs and store them locally*)
	Output_Params[1]:=Velocity_Percentage;
	Output_Params[2]:=0;
	Output_Params[3]:=0;
	Output_Params[4]:=0;
	Output_Params[5]:=0;
	Output_Params[6]:=0;

	(* If Values have change, Reinitialise Outputs*)

	IF FirstScan=0 OR 
		Robot.Outputs.MotionCommand.MoveSubIndex001 <> Output_Params[1] OR 
		Robot.Outputs.MotionCommand.MoveSubIndex002 <> Output_Params[2] OR 
		Robot.Outputs.MotionCommand.MoveSubIndex003 <> Output_Params[3] OR
		Robot.Outputs.MotionCommand.MoveSubIndex004 <> Output_Params[4] OR 
		Robot.Outputs.MotionCommand.MoveSubIndex005 <> Output_Params[5] OR 
		Robot.Outputs.MotionCommand.MoveSubIndex006 <> Output_Params[6] 
	THEN
		Buffered := FALSE;
		Sent := FALSE;
	END_IF;


	(*if not in legacy mode, Act Setpoint*)
	IF Robot.Outputs.MotionControl.MoveID <> 0 THEN
	    Robot.Outputs.MotionControl.SetPoint := TRUE;
	END_IF;

	(* To send _Move, send _Move ID *)
	IF NOT Buffered AND NOT Sent THEN
	    
	    Robot.Outputs.MotionCommand.MoveCommand	:= EnumToNum(Meca500Cmd#SetJointVel);
	    Robot.Outputs.MotionCommand.MoveSubIndex001 := Output_Params[1];
		Robot.Outputs.MotionCommand.MoveSubIndex002 := Output_Params[2];
		Robot.Outputs.MotionCommand.MoveSubIndex003 := Output_Params[3];
		Robot.Outputs.MotionCommand.MoveSubIndex004 := Output_Params[4];
		Robot.Outputs.MotionCommand.MoveSubIndex005 := Output_Params[5];
		Robot.Outputs.MotionCommand.MoveSubIndex006 := Output_Params[6];
	    
	    IF ExternalStateControl THEN
	        IF ExternalMoveID <> 0 AND ExternalMoveID <> 32080 AND ExternalMoveID <> 32081 THEN
	            Robot.Outputs.MotionControl.MoveID := ExternalMoveID;
	            Sent := TRUE;
	        END_IF;
	        
	    ELSE (*Not External Control*)
	        IF Robot.Outputs.MotionControl.MoveID = 32080 THEN
	            Robot.Outputs.MotionControl.MoveID := 32081;
	        ELSIF Robot.Outputs.MotionControl.MoveID = 32081 THEN
	            Robot.Outputs.MotionControl.MoveID := 32080;
	        ELSIF Robot.Outputs.MotionControl.MoveID <> 32080 OR Robot.Outputs.MotionControl.MoveID <> 32081 THEN
	            Robot.Outputs.MotionControl.MoveID := 32080;
	        END_IF;
	        Sent := TRUE;
	    END_IF;
	END_IF;

	(* Check if command has been sent, if so, check if it was received *)
	IF Sent AND
	    Robot.Outputs.MotionCommand.MoveCommand = EnumToNum(Meca500Cmd#SetJointVel) AND
	    Robot.Outputs.MotionCommand.MoveSubIndex001 = Output_Params[1] AND 
		Robot.Outputs.MotionCommand.MoveSubIndex002 = Output_Params[2] AND 
		Robot.Outputs.MotionCommand.MoveSubIndex003 = Output_Params[3] AND 
		Robot.Outputs.MotionCommand.MoveSubIndex004 = Output_Params[4] AND 
		Robot.Outputs.MotionCommand.MoveSubIndex005 = Output_Params[5] AND 
		Robot.Outputs.MotionCommand.MoveSubIndex006 = Output_Params[6] AND
		Robot.Inputs.Motion.MoveID = Robot.Outputs.MotionControl.MoveID 
	THEN
		 Buffered := TRUE;
	END_IF;


	(*If External _Move ID is equal to Internal, raise an error*)
	IF ExternalMoveID = 32080 OR ExternalMoveID = 32081 THEN
	    Error := TRUE;
	END_IF;

	FirstScan := TRUE;
ELSE
	FirstScan := False;
	Sent := FALSE;
	Buffered := FALSE;
END_IF;
END_FUNCTION_BLOCK

FUNCTION_BLOCK Meca500_SetTorqueLimitCfg
VAR
    Output_Params : array[1..6] of real;
    FirstScan : BOOL := False;
END_VAR
VAR_INPUT
    Execute : BOOL;
    Severity : REAL;
    Mode : REAL;
END_VAR
VAR_OUTPUT
    Sent : BOOL;
    Buffered : BOOL;
    Error : BOOL;
END_VAR
VAR_IN_OUT
    Robot : Meca500;
END_VAR
VAR_INPUT
    ExternalStateControl : BOOL;
    ExternalMoveID : UINT;
END_VAR
IF Execute THEN	
	(*Collect Inputs and store them locally*)
	Output_Params[1]:=Severity;
	Output_Params[2]:=Mode;
	Output_Params[3]:=0;
	Output_Params[4]:=0;
	Output_Params[5]:=0;
	Output_Params[6]:=0;

	(* If Values have change, Reinitialise Outputs*)

	IF FirstScan=0 OR 
		Robot.Outputs.MotionCommand.MoveSubIndex001 <> Output_Params[1] OR 
		Robot.Outputs.MotionCommand.MoveSubIndex002 <> Output_Params[2] OR 
		Robot.Outputs.MotionCommand.MoveSubIndex003 <> Output_Params[3] OR
		Robot.Outputs.MotionCommand.MoveSubIndex004 <> Output_Params[4] OR 
		Robot.Outputs.MotionCommand.MoveSubIndex005 <> Output_Params[5] OR 
		Robot.Outputs.MotionCommand.MoveSubIndex006 <> Output_Params[6] 
	THEN
		Buffered := FALSE;
		Sent := FALSE;
	END_IF;


	(*if not in legacy mode, Act Setpoint*)
	IF Robot.Outputs.MotionControl.MoveID <> 0 THEN
	    Robot.Outputs.MotionControl.SetPoint := TRUE;
	END_IF;

	(* To send _Move, send _Move ID *)
	IF NOT Buffered AND NOT Sent THEN
	    
	    Robot.Outputs.MotionCommand.MoveCommand	:= EnumToNum(Meca500Cmd#SetTorquesLimitCfg);
	    Robot.Outputs.MotionCommand.MoveSubIndex001 := Output_Params[1];
		Robot.Outputs.MotionCommand.MoveSubIndex002 := Output_Params[2];
		Robot.Outputs.MotionCommand.MoveSubIndex003 := Output_Params[3];
		Robot.Outputs.MotionCommand.MoveSubIndex004 := Output_Params[4];
		Robot.Outputs.MotionCommand.MoveSubIndex005 := Output_Params[5];
		Robot.Outputs.MotionCommand.MoveSubIndex006 := Output_Params[6];
	    
	    IF ExternalStateControl THEN
	        IF ExternalMoveID <> 0 AND ExternalMoveID <> 32280 AND ExternalMoveID <> 32281 THEN
	            Robot.Outputs.MotionControl.MoveID := ExternalMoveID;
	            Sent := TRUE;
	        END_IF;
	        
	    ELSE (*Not External Control*)
	        IF Robot.Outputs.MotionControl.MoveID = 32280 THEN
	            Robot.Outputs.MotionControl.MoveID := 32281;
	        ELSIF Robot.Outputs.MotionControl.MoveID = 32281 THEN
	            Robot.Outputs.MotionControl.MoveID := 32280;
	        ELSIF Robot.Outputs.MotionControl.MoveID <> 32280 OR Robot.Outputs.MotionControl.MoveID <> 32281 THEN
	            Robot.Outputs.MotionControl.MoveID := 32280;
	        END_IF;
	        Sent := TRUE;
	    END_IF;
	END_IF;

	(* Check if command has been sent, if so, check if it was received *)
	IF Sent AND
	    Robot.Outputs.MotionCommand.MoveCommand = EnumToNum(Meca500Cmd#SetTorquesLimitCfg) AND
	    Robot.Outputs.MotionCommand.MoveSubIndex001 = Output_Params[1] AND 
		Robot.Outputs.MotionCommand.MoveSubIndex002 = Output_Params[2] AND 
		Robot.Outputs.MotionCommand.MoveSubIndex003 = Output_Params[3] AND 
		Robot.Outputs.MotionCommand.MoveSubIndex004 = Output_Params[4] AND 
		Robot.Outputs.MotionCommand.MoveSubIndex005 = Output_Params[5] AND 
		Robot.Outputs.MotionCommand.MoveSubIndex006 = Output_Params[6] AND
		Robot.Inputs.Motion.MoveID = Robot.Outputs.MotionControl.MoveID 
	THEN
		 Buffered := TRUE;
	END_IF;


	(*If External _Move ID is equal to Internal, raise an error*)
	IF ExternalMoveID = 32280 OR ExternalMoveID = 32281 THEN
	    Error := TRUE;
	END_IF;

	FirstScan := TRUE;
ELSE
	FirstScan := False;
	Sent := FALSE;
	Buffered := FALSE;
END_IF;
END_FUNCTION_BLOCK

FUNCTION_BLOCK Meca500_SetTorqueLimits
VAR
    Output_Params : array[1..6] of real;
    FirstScan : BOOL := False;
END_VAR
VAR_INPUT
    Execute : BOOL;
    Joint_1_Limit : REAL;
    Joint_2_Limit : REAL;
    Joint_3_Limit : REAL;
    Joint_4_Limit : REAL;
    Joint_5_Limit : REAL;
    Joint_6_Limit : REAL;
END_VAR
VAR_OUTPUT
    Sent : BOOL;
    Buffered : BOOL;
    Error : BOOL;
END_VAR
VAR_IN_OUT
    Robot : Meca500;
END_VAR
VAR_INPUT
    ExternalStateControl : BOOL;
    ExternalMoveID : UINT;
END_VAR
IF Execute THEN	
	(*Collect Inputs and store them locally*)
	Output_Params[1]:=Joint_1_Limit;
	Output_Params[2]:=Joint_2_Limit;
	Output_Params[3]:=Joint_3_Limit;
	Output_Params[4]:=Joint_4_Limit;
	Output_Params[5]:=Joint_5_Limit;
	Output_Params[6]:=Joint_6_Limit;


	(* If Values have change, Reinitialise Outputs*)

	IF FirstScan=0 OR 
		Robot.Outputs.MotionCommand.MoveSubIndex001 <> Output_Params[1] OR 
		Robot.Outputs.MotionCommand.MoveSubIndex002 <> Output_Params[2] OR 
		Robot.Outputs.MotionCommand.MoveSubIndex003 <> Output_Params[3] OR
		Robot.Outputs.MotionCommand.MoveSubIndex004 <> Output_Params[4] OR 
		Robot.Outputs.MotionCommand.MoveSubIndex005 <> Output_Params[5] OR 
		Robot.Outputs.MotionCommand.MoveSubIndex006 <> Output_Params[6] 
	THEN
		Buffered := FALSE;
		Sent := FALSE;
	END_IF;


	(*if not in legacy mode, Act Setpoint*)
	IF Robot.Outputs.MotionControl.MoveID <> 0 THEN
	    Robot.Outputs.MotionControl.SetPoint := TRUE;
	END_IF;

	(* To send _Move, send _Move ID *)
	IF NOT Buffered AND NOT Sent THEN
	    
	    Robot.Outputs.MotionCommand.MoveCommand	:= EnumToNum(Meca500Cmd#SetTorqueLimits);
	    Robot.Outputs.MotionCommand.MoveSubIndex001 := Output_Params[1];
		Robot.Outputs.MotionCommand.MoveSubIndex002 := Output_Params[2];
		Robot.Outputs.MotionCommand.MoveSubIndex003 := Output_Params[3];
		Robot.Outputs.MotionCommand.MoveSubIndex004 := Output_Params[4];
		Robot.Outputs.MotionCommand.MoveSubIndex005 := Output_Params[5];
		Robot.Outputs.MotionCommand.MoveSubIndex006 := Output_Params[6];
	    
	    IF ExternalStateControl THEN
	        IF ExternalMoveID <> 0 AND ExternalMoveID <> 32270 AND ExternalMoveID <> 32271 THEN
	            Robot.Outputs.MotionControl.MoveID := ExternalMoveID;
	            Sent := TRUE;
	        END_IF;
	        
	    ELSE (*Not External Control*)
	        IF Robot.Outputs.MotionControl.MoveID = 32270 THEN
	            Robot.Outputs.MotionControl.MoveID := 32271;
	        ELSIF Robot.Outputs.MotionControl.MoveID = 32271 THEN
	            Robot.Outputs.MotionControl.MoveID := 32270;
	        ELSIF Robot.Outputs.MotionControl.MoveID <> 32270 OR Robot.Outputs.MotionControl.MoveID <> 32271 THEN
	            Robot.Outputs.MotionControl.MoveID := 32270;
	        END_IF;
	        Sent := TRUE;
	    END_IF;
	END_IF;

	(* Check if command has been sent, if so, check if it was received *)
	IF Sent AND
	    Robot.Outputs.MotionCommand.MoveCommand = EnumToNum(Meca500Cmd#SetTorqueLimits) AND
	    Robot.Outputs.MotionCommand.MoveSubIndex001 = Output_Params[1] AND 
		Robot.Outputs.MotionCommand.MoveSubIndex002 = Output_Params[2] AND 
		Robot.Outputs.MotionCommand.MoveSubIndex003 = Output_Params[3] AND 
		Robot.Outputs.MotionCommand.MoveSubIndex004 = Output_Params[4] AND 
		Robot.Outputs.MotionCommand.MoveSubIndex005 = Output_Params[5] AND 
		Robot.Outputs.MotionCommand.MoveSubIndex006 = Output_Params[6] AND
		Robot.Inputs.Motion.MoveID = Robot.Outputs.MotionControl.MoveID 
	THEN
		 Buffered := TRUE;
	END_IF;


	(*If External _Move ID is equal to Internal, raise an error*)
	IF ExternalMoveID = 32270 OR ExternalMoveID = 32271 THEN
	    Error := TRUE;
	END_IF;

	FirstScan := TRUE;
ELSE
	FirstScan := False;
	Sent := FALSE;
	Buffered := FALSE;
END_IF;
END_FUNCTION_BLOCK

FUNCTION_BLOCK Meca500_SetTrf
VAR
    Output_Params : array[1..6] of real;
    FirstScan : BOOL := False;
END_VAR
VAR_INPUT
    Execute : BOOL;
    Pose_X_Pos : REAL;
    Pose_Y_Pos : REAL;
    Pose_Z_Pos : REAL;
    Pose_rX_Angle : REAL;
    Pose_rY_Angle : REAL;
    Pose_rZ_Angle : REAL;
END_VAR
VAR_OUTPUT
    Sent : BOOL;
    Buffered : BOOL;
    Error : BOOL;
END_VAR
VAR_IN_OUT
    Robot : Meca500;
END_VAR
VAR_INPUT
    ExternalStateControl : BOOL;
    ExternalMoveID : UINT;
END_VAR
IF Execute THEN	
	(*Collect Inputs and store them locally*)
	Output_Params[1]:=Pose_X_Pos;
	Output_Params[2]:=Pose_Y_Pos;
	Output_Params[3]:=Pose_Z_Pos;
	Output_Params[4]:=Pose_rX_Angle;
	Output_Params[5]:=Pose_rY_Angle;
	Output_Params[6]:=Pose_rZ_Angle;

	(* If Values have change, Reinitialise Outputs*)

	IF FirstScan=0 OR 
		Robot.Outputs.MotionCommand.MoveSubIndex001 <> Output_Params[1] OR 
		Robot.Outputs.MotionCommand.MoveSubIndex002 <> Output_Params[2] OR 
		Robot.Outputs.MotionCommand.MoveSubIndex003 <> Output_Params[3] OR
		Robot.Outputs.MotionCommand.MoveSubIndex004 <> Output_Params[4] OR 
		Robot.Outputs.MotionCommand.MoveSubIndex005 <> Output_Params[5] OR 
		Robot.Outputs.MotionCommand.MoveSubIndex006 <> Output_Params[6] 
	THEN
		Buffered := FALSE;
		Sent := FALSE;
	END_IF;


	(*if not in legacy mode, Act Setpoint*)
	IF Robot.Outputs.MotionControl.MoveID <> 0 THEN
	    Robot.Outputs.MotionControl.SetPoint := TRUE;
	END_IF;

	(* To send _Move, send _Move ID *)
	IF NOT Buffered AND NOT Sent THEN
	    
	    Robot.Outputs.MotionCommand.MoveCommand	:= EnumToNum(Meca500Cmd#SetTrf);
	    Robot.Outputs.MotionCommand.MoveSubIndex001 := Output_Params[1];
		Robot.Outputs.MotionCommand.MoveSubIndex002 := Output_Params[2];
		Robot.Outputs.MotionCommand.MoveSubIndex003 := Output_Params[3];
		Robot.Outputs.MotionCommand.MoveSubIndex004 := Output_Params[4];
		Robot.Outputs.MotionCommand.MoveSubIndex005 := Output_Params[5];
		Robot.Outputs.MotionCommand.MoveSubIndex006 := Output_Params[6];
	    
	    IF ExternalStateControl THEN
	        IF ExternalMoveID <> 0 AND ExternalMoveID <> 32130 AND ExternalMoveID <> 32131 THEN
	            Robot.Outputs.MotionControl.MoveID := ExternalMoveID;
	            Sent := TRUE;
	        END_IF;
	        
	    ELSE (*Not External Control*)
	        IF Robot.Outputs.MotionControl.MoveID = 32130 THEN
	            Robot.Outputs.MotionControl.MoveID := 32131;
	        ELSIF Robot.Outputs.MotionControl.MoveID = 32131 THEN
	            Robot.Outputs.MotionControl.MoveID := 32130;
	        ELSIF Robot.Outputs.MotionControl.MoveID <> 32130 OR Robot.Outputs.MotionControl.MoveID <> 32131 THEN
	            Robot.Outputs.MotionControl.MoveID := 32130;
	        END_IF;
	        Sent := TRUE;
	    END_IF;
	END_IF;

	(* Check if command has been sent, if so, check if it was received *)
	IF Sent AND
	    Robot.Outputs.MotionCommand.MoveCommand = EnumToNum(Meca500Cmd#SetTrf) AND
	    Robot.Outputs.MotionCommand.MoveSubIndex001 = Output_Params[1] AND 
		Robot.Outputs.MotionCommand.MoveSubIndex002 = Output_Params[2] AND 
		Robot.Outputs.MotionCommand.MoveSubIndex003 = Output_Params[3] AND 
		Robot.Outputs.MotionCommand.MoveSubIndex004 = Output_Params[4] AND 
		Robot.Outputs.MotionCommand.MoveSubIndex005 = Output_Params[5] AND 
		Robot.Outputs.MotionCommand.MoveSubIndex006 = Output_Params[6] AND
		Robot.Inputs.Motion.MoveID = Robot.Outputs.MotionControl.MoveID 
	THEN
		 Buffered := TRUE;
	END_IF;


	(*If External _Move ID is equal to Internal, raise an error*)
	IF ExternalMoveID = 32130 OR ExternalMoveID = 32131 THEN
	    Error := TRUE;
	END_IF;

	FirstScan := TRUE;
ELSE
	FirstScan := False;
	Sent := FALSE;
	Buffered := FALSE;
END_IF;
END_FUNCTION_BLOCK

FUNCTION_BLOCK Meca500_SetValveState
VAR
    Output_Params : array[1..6] of real;
    FirstScan : BOOL := False;
END_VAR
VAR_INPUT
    Execute : BOOL;
    V1 : REAL;
    V2 : REAL;
END_VAR
VAR_OUTPUT
    Sent : BOOL;
    Buffered : BOOL;
    Error : BOOL;
END_VAR
VAR_IN_OUT
    Robot : Meca500;
END_VAR
VAR_INPUT
    ExternalStateControl : BOOL;
    ExternalMoveID : UINT;
END_VAR
IF Execute THEN	
	(*Collect Inputs and store them locally*)
	Output_Params[1]:=V1;
	Output_Params[2]:=V2;
	Output_Params[3]:=0;
	Output_Params[4]:=0;
	Output_Params[5]:=0;
	Output_Params[6]:=0;

	(* If Values have change, Reinitialise Outputs*)

	IF FirstScan=0 OR 
		Robot.Outputs.MotionCommand.MoveSubIndex001 <> Output_Params[1] OR 
		Robot.Outputs.MotionCommand.MoveSubIndex002 <> Output_Params[2] OR 
		Robot.Outputs.MotionCommand.MoveSubIndex003 <> Output_Params[3] OR
		Robot.Outputs.MotionCommand.MoveSubIndex004 <> Output_Params[4] OR 
		Robot.Outputs.MotionCommand.MoveSubIndex005 <> Output_Params[5] OR 
		Robot.Outputs.MotionCommand.MoveSubIndex006 <> Output_Params[6] 
	THEN
		Buffered := FALSE;
		Sent := FALSE;
	END_IF;


	(*if not in legacy mode, Act Setpoint*)
	IF Robot.Outputs.MotionControl.MoveID <> 0 THEN
	    Robot.Outputs.MotionControl.SetPoint := TRUE;
	END_IF;

	(* To send _Move, send _Move ID *)
	IF NOT Buffered AND NOT Sent THEN
	    
	    Robot.Outputs.MotionCommand.MoveCommand	:= EnumToNum(Meca500Cmd#SetValveState);
	    Robot.Outputs.MotionCommand.MoveSubIndex001 := Output_Params[1];
		Robot.Outputs.MotionCommand.MoveSubIndex002 := Output_Params[2];
		Robot.Outputs.MotionCommand.MoveSubIndex003 := Output_Params[3];
		Robot.Outputs.MotionCommand.MoveSubIndex004 := Output_Params[4];
		Robot.Outputs.MotionCommand.MoveSubIndex005 := Output_Params[5];
		Robot.Outputs.MotionCommand.MoveSubIndex006 := Output_Params[6];
	    
	    IF ExternalStateControl THEN
	        IF ExternalMoveID <> 0 AND ExternalMoveID <> 32300 AND ExternalMoveID <> 32301 THEN
	            Robot.Outputs.MotionControl.MoveID := ExternalMoveID;
	            Sent := TRUE;
	        END_IF;
	        
	    ELSE (*Not External Control*)
	        IF Robot.Outputs.MotionControl.MoveID = 32300 THEN
	            Robot.Outputs.MotionControl.MoveID := 32301;
	        ELSIF Robot.Outputs.MotionControl.MoveID = 32301 THEN
	            Robot.Outputs.MotionControl.MoveID := 32300;
	        ELSIF Robot.Outputs.MotionControl.MoveID <> 32300 OR Robot.Outputs.MotionControl.MoveID <> 32301 THEN
	            Robot.Outputs.MotionControl.MoveID := 32300;
	        END_IF;
	        Sent := TRUE;
	    END_IF;
	END_IF;

	(* Check if command has been sent, if so, check if it was received *)
	IF Sent AND
	    Robot.Outputs.MotionCommand.MoveCommand = EnumToNum(Meca500Cmd#SetValveState) AND
	    Robot.Outputs.MotionCommand.MoveSubIndex001 = Output_Params[1] AND 
		Robot.Outputs.MotionCommand.MoveSubIndex002 = Output_Params[2] AND 
		Robot.Outputs.MotionCommand.MoveSubIndex003 = Output_Params[3] AND 
		Robot.Outputs.MotionCommand.MoveSubIndex004 = Output_Params[4] AND 
		Robot.Outputs.MotionCommand.MoveSubIndex005 = Output_Params[5] AND 
		Robot.Outputs.MotionCommand.MoveSubIndex006 = Output_Params[6] AND
		Robot.Inputs.Motion.MoveID = Robot.Outputs.MotionControl.MoveID 
	THEN
		 Buffered := TRUE;
	END_IF;


	(*If External _Move ID is equal to Internal, raise an error*)
	IF ExternalMoveID = 32300 OR ExternalMoveID = 32301 THEN
	    Error := TRUE;
	END_IF;

	FirstScan := TRUE;
ELSE
	FirstScan := False;
	Sent := FALSE;
	Buffered := FALSE;
END_IF;
END_FUNCTION_BLOCK

FUNCTION_BLOCK Meca500_SetVelTimeout
VAR
    Output_Params : array[1..6] of real;
    FirstScan : BOOL := False;
END_VAR
VAR_INPUT
    Execute : BOOL;
    Seconds : REAL;
END_VAR
VAR_OUTPUT
    Sent : BOOL;
    Buffered : BOOL;
    Error : BOOL;
END_VAR
VAR_IN_OUT
    Robot : Meca500;
END_VAR
VAR_INPUT
    ExternalStateControl : BOOL;
    ExternalMoveID : UINT;
END_VAR
IF Execute THEN	
	(*Collect Inputs and store them locally*)
	Output_Params[1]:=Seconds;
	Output_Params[2]:=0;
	Output_Params[3]:=0;
	Output_Params[4]:=0;
	Output_Params[5]:=0;
	Output_Params[6]:=0;


	(* If Values have change, Reinitialise Outputs*)

	IF FirstScan=0 OR 
		Robot.Outputs.MotionCommand.MoveSubIndex001 <> Output_Params[1] OR 
		Robot.Outputs.MotionCommand.MoveSubIndex002 <> Output_Params[2] OR 
		Robot.Outputs.MotionCommand.MoveSubIndex003 <> Output_Params[3] OR
		Robot.Outputs.MotionCommand.MoveSubIndex004 <> Output_Params[4] OR 
		Robot.Outputs.MotionCommand.MoveSubIndex005 <> Output_Params[5] OR 
		Robot.Outputs.MotionCommand.MoveSubIndex006 <> Output_Params[6] 
	THEN
		Buffered := FALSE;
		Sent := FALSE;
	END_IF;


	(*if not in legacy mode, Act Setpoint*)
	IF Robot.Outputs.MotionControl.MoveID <> 0 THEN
	    Robot.Outputs.MotionControl.SetPoint := TRUE;
	END_IF;

	(* To send _Move, send _Move ID *)
	IF NOT Buffered AND NOT Sent THEN
	    
	    Robot.Outputs.MotionCommand.MoveCommand	:= EnumToNum(Meca500Cmd#SetVelTimeout);
	    Robot.Outputs.MotionCommand.MoveSubIndex001 := Output_Params[1];
		Robot.Outputs.MotionCommand.MoveSubIndex002 := Output_Params[2];
		Robot.Outputs.MotionCommand.MoveSubIndex003 := Output_Params[3];
		Robot.Outputs.MotionCommand.MoveSubIndex004 := Output_Params[4];
		Robot.Outputs.MotionCommand.MoveSubIndex005 := Output_Params[5];
		Robot.Outputs.MotionCommand.MoveSubIndex006 := Output_Params[6];
	    
	    IF ExternalStateControl THEN
	        IF ExternalMoveID <> 0 AND ExternalMoveID <> 32240 AND ExternalMoveID <> 32241 THEN
	            Robot.Outputs.MotionControl.MoveID := ExternalMoveID;
	            Sent := TRUE;
	        END_IF;
	        
	    ELSE (*Not External Control*)
	        IF Robot.Outputs.MotionControl.MoveID = 32240 THEN
	            Robot.Outputs.MotionControl.MoveID := 32241;
	        ELSIF Robot.Outputs.MotionControl.MoveID = 32241 THEN
	            Robot.Outputs.MotionControl.MoveID := 32240;
	        ELSIF Robot.Outputs.MotionControl.MoveID <> 32240 OR Robot.Outputs.MotionControl.MoveID <> 32241 THEN
	            Robot.Outputs.MotionControl.MoveID := 32240;
	        END_IF;
	        Sent := TRUE;
	    END_IF;
	END_IF;

	(* Check if command has been sent, if so, check if it was received *)
	IF Sent AND
	    Robot.Outputs.MotionCommand.MoveCommand = EnumToNum(Meca500Cmd#SetVelTimeout) AND
	    Robot.Outputs.MotionCommand.MoveSubIndex001 = Output_Params[1] AND 
		Robot.Outputs.MotionCommand.MoveSubIndex002 = Output_Params[2] AND 
		Robot.Outputs.MotionCommand.MoveSubIndex003 = Output_Params[3] AND 
		Robot.Outputs.MotionCommand.MoveSubIndex004 = Output_Params[4] AND 
		Robot.Outputs.MotionCommand.MoveSubIndex005 = Output_Params[5] AND 
		Robot.Outputs.MotionCommand.MoveSubIndex006 = Output_Params[6] AND
		Robot.Inputs.Motion.MoveID = Robot.Outputs.MotionControl.MoveID 
	THEN
		 Buffered := TRUE;
	END_IF;


	(*If External _Move ID is equal to Internal, raise an error*)
	IF ExternalMoveID = 32240 OR ExternalMoveID = 32241 THEN
	    Error := TRUE;
	END_IF;

	FirstScan := TRUE;
ELSE
	FirstScan := False;
	Sent := FALSE;
	Buffered := FALSE;
END_IF;
END_FUNCTION_BLOCK

FUNCTION_BLOCK Meca500_SetWrf
VAR
    Output_Params : array[1..6] of real;
    FirstScan : BOOL := False;
END_VAR
VAR_INPUT
    Execute : BOOL;
    Pose_X_Pos : REAL;
    Pose_Y_Pos : REAL;
    Pose_Z_Pos : REAL;
    Pose_rX_Angle : REAL;
    Pose_rY_Angle : REAL;
    Pose_rZ_Angle : REAL;
END_VAR
VAR_OUTPUT
    Sent : BOOL;
    Buffered : BOOL;
    Error : BOOL;
END_VAR
VAR_IN_OUT
    Robot : Meca500;
END_VAR
VAR_INPUT
    ExternalStateControl : BOOL;
    ExternalMoveID : UINT;
END_VAR
IF Execute THEN	
	(*Collect Inputs and store them locally*)
	Output_Params[1]:=Pose_X_Pos;
	Output_Params[2]:=Pose_Y_Pos;
	Output_Params[3]:=Pose_Z_Pos;
	Output_Params[4]:=Pose_rX_Angle;
	Output_Params[5]:=Pose_rY_Angle;
	Output_Params[6]:=Pose_rZ_Angle;

	(* If Values have change, Reinitialise Outputs*)

	IF FirstScan=0 OR 
		Robot.Outputs.MotionCommand.MoveSubIndex001 <> Output_Params[1] OR 
		Robot.Outputs.MotionCommand.MoveSubIndex002 <> Output_Params[2] OR 
		Robot.Outputs.MotionCommand.MoveSubIndex003 <> Output_Params[3] OR
		Robot.Outputs.MotionCommand.MoveSubIndex004 <> Output_Params[4] OR 
		Robot.Outputs.MotionCommand.MoveSubIndex005 <> Output_Params[5] OR 
		Robot.Outputs.MotionCommand.MoveSubIndex006 <> Output_Params[6] 
	THEN
		Buffered := FALSE;
		Sent := FALSE;
	END_IF;


	(*if not in legacy mode, Act Setpoint*)
	IF Robot.Outputs.MotionControl.MoveID <> 0 THEN
	    Robot.Outputs.MotionControl.SetPoint := TRUE;
	END_IF;

	(* To send _Move, send _Move ID *)
	IF NOT Buffered AND NOT Sent THEN
	    
	    Robot.Outputs.MotionCommand.MoveCommand	:= EnumToNum(Meca500Cmd#SetWrf);
	    Robot.Outputs.MotionCommand.MoveSubIndex001 := Output_Params[1];
		Robot.Outputs.MotionCommand.MoveSubIndex002 := Output_Params[2];
		Robot.Outputs.MotionCommand.MoveSubIndex003 := Output_Params[3];
		Robot.Outputs.MotionCommand.MoveSubIndex004 := Output_Params[4];
		Robot.Outputs.MotionCommand.MoveSubIndex005 := Output_Params[5];
		Robot.Outputs.MotionCommand.MoveSubIndex006 := Output_Params[6];
	    
	    IF ExternalStateControl THEN
	        IF ExternalMoveID <> 0 AND ExternalMoveID <> 32140 AND ExternalMoveID <> 32141 THEN
	            Robot.Outputs.MotionControl.MoveID := ExternalMoveID;
	            Sent := TRUE;
	        END_IF;
	        
	    ELSE (*Not External Control*)
	        IF Robot.Outputs.MotionControl.MoveID = 32140 THEN
	            Robot.Outputs.MotionControl.MoveID := 32141;
	        ELSIF Robot.Outputs.MotionControl.MoveID = 32141 THEN
	            Robot.Outputs.MotionControl.MoveID := 32140;
	        ELSIF Robot.Outputs.MotionControl.MoveID <> 32140 OR Robot.Outputs.MotionControl.MoveID <> 32141 THEN
	            Robot.Outputs.MotionControl.MoveID := 32140;
	        END_IF;
	        Sent := TRUE;
	    END_IF;
	END_IF;

	(* Check if command has been sent, if so, check if it was received *)
	IF Sent AND
	    Robot.Outputs.MotionCommand.MoveCommand = EnumToNum(Meca500Cmd#SetWrf) AND
	    Robot.Outputs.MotionCommand.MoveSubIndex001 = Output_Params[1] AND 
		Robot.Outputs.MotionCommand.MoveSubIndex002 = Output_Params[2] AND 
		Robot.Outputs.MotionCommand.MoveSubIndex003 = Output_Params[3] AND 
		Robot.Outputs.MotionCommand.MoveSubIndex004 = Output_Params[4] AND 
		Robot.Outputs.MotionCommand.MoveSubIndex005 = Output_Params[5] AND 
		Robot.Outputs.MotionCommand.MoveSubIndex006 = Output_Params[6] AND
		Robot.Inputs.Motion.MoveID = Robot.Outputs.MotionControl.MoveID 
	THEN
		 Buffered := TRUE;
	END_IF;


	(*If External _Move ID is equal to Internal, raise an error*)
	IF ExternalMoveID = 32140 OR ExternalMoveID = 32141 THEN
	    Error := TRUE;
	END_IF;

	FirstScan := TRUE;
ELSE
	FirstScan := False;
	Sent := FALSE;
	Buffered := FALSE;
END_IF;
END_FUNCTION_BLOCK

FUNCTION_BLOCK Meca500_StartProgram
VAR
    Output_Params : array[1..6] of real;
    FirstScan : BOOL := False;
END_VAR
VAR_INPUT
    Execute : BOOL;
    n : REAL;
END_VAR
VAR_OUTPUT
    Sent : BOOL;
    Buffered : BOOL;
    Error : BOOL;
END_VAR
VAR_IN_OUT
    Robot : Meca500;
END_VAR
VAR_INPUT
    ExternalStateControl : BOOL;
    ExternalMoveID : UINT;
END_VAR
IF Execute THEN	
	(*Collect Inputs and store them locally*)
	Output_Params[1]:=n;
	Output_Params[2]:=0;
	Output_Params[3]:=0;
	Output_Params[4]:=0;
	Output_Params[5]:=0;
	Output_Params[6]:=0;


	(* If Values have change, Reinitialise Outputs*)

	IF FirstScan=0 OR 
		Robot.Outputs.MotionCommand.MoveSubIndex001 <> Output_Params[1] OR 
		Robot.Outputs.MotionCommand.MoveSubIndex002 <> Output_Params[2] OR 
		Robot.Outputs.MotionCommand.MoveSubIndex003 <> Output_Params[3] OR
		Robot.Outputs.MotionCommand.MoveSubIndex004 <> Output_Params[4] OR 
		Robot.Outputs.MotionCommand.MoveSubIndex005 <> Output_Params[5] OR 
		Robot.Outputs.MotionCommand.MoveSubIndex006 <> Output_Params[6] 
	THEN
		Buffered := FALSE;
		Sent := FALSE;
	END_IF;


	(*if not in legacy mode, Act Setpoint*)
	IF Robot.Outputs.MotionControl.MoveID <> 0 THEN
	    Robot.Outputs.MotionControl.SetPoint := TRUE;
	END_IF;

	(* To send _Move, send _Move ID *)
	IF NOT Buffered AND NOT Sent THEN
	    
	    Robot.Outputs.MotionCommand.MoveCommand	:= EnumToNum(Meca500Cmd#StartProgram);
	    Robot.Outputs.MotionCommand.MoveSubIndex001 := Output_Params[1];
		Robot.Outputs.MotionCommand.MoveSubIndex002 := Output_Params[2];
		Robot.Outputs.MotionCommand.MoveSubIndex003 := Output_Params[3];
		Robot.Outputs.MotionCommand.MoveSubIndex004 := Output_Params[4];
		Robot.Outputs.MotionCommand.MoveSubIndex005 := Output_Params[5];
		Robot.Outputs.MotionCommand.MoveSubIndex006 := Output_Params[6];
	    
	    IF ExternalStateControl THEN
	        IF ExternalMoveID <> 0 AND ExternalMoveID <> 31900 AND ExternalMoveID <> 31901 THEN
	            Robot.Outputs.MotionControl.MoveID := ExternalMoveID;
	            Sent := TRUE;
	        END_IF;
	        
	    ELSE (*Not External Control*)
	        IF Robot.Outputs.MotionControl.MoveID = 31900 THEN
	            Robot.Outputs.MotionControl.MoveID := 31901;
	        ELSIF Robot.Outputs.MotionControl.MoveID = 31901 THEN
	            Robot.Outputs.MotionControl.MoveID := 31900;
	        ELSIF Robot.Outputs.MotionControl.MoveID <> 31900 OR Robot.Outputs.MotionControl.MoveID <> 31901 THEN
	            Robot.Outputs.MotionControl.MoveID := 31900;
	        END_IF;
	        Sent := TRUE;
	    END_IF;
	END_IF;

	(* Check if command has been sent, if so, check if it was received *)
	IF Sent AND
	    Robot.Outputs.MotionCommand.MoveCommand = EnumToNum(Meca500Cmd#StartProgram) AND
	    Robot.Outputs.MotionCommand.MoveSubIndex001 = Output_Params[1] AND 
		Robot.Outputs.MotionCommand.MoveSubIndex002 = Output_Params[2] AND 
		Robot.Outputs.MotionCommand.MoveSubIndex003 = Output_Params[3] AND 
		Robot.Outputs.MotionCommand.MoveSubIndex004 = Output_Params[4] AND 
		Robot.Outputs.MotionCommand.MoveSubIndex005 = Output_Params[5] AND 
		Robot.Outputs.MotionCommand.MoveSubIndex006 = Output_Params[6] AND
		Robot.Inputs.Motion.MoveID = Robot.Outputs.MotionControl.MoveID 
	THEN
		 Buffered := TRUE;
	END_IF;


	(*If External _Move ID is equal to Internal, raise an error*)
	IF ExternalMoveID = 31900 OR ExternalMoveID = 31901 THEN
	    Error := TRUE;
	END_IF;

	FirstScan := TRUE;
ELSE
	FirstScan := False;
	Buffered := FALSE;
		Sent := FALSE;
END_IF;
END_FUNCTION_BLOCK

FUNCTION_BLOCK Meca500_SetJointVelLimit
VAR
    Output_Params : array[1..6] of real;
    FirstScan : BOOL := False;
END_VAR
VAR_INPUT
    Execute : BOOL;
    MaxJointVel : REAL;
END_VAR
VAR_OUTPUT
    Sent : BOOL;
    Buffered : BOOL;
    Error : BOOL;
END_VAR
VAR_IN_OUT
    Robot : Meca500;
END_VAR
VAR_INPUT
    ExternalStateControl : BOOL;
    ExternalMoveID : UINT;
END_VAR
IF Execute THEN	
	(*Collect Inputs and store them locally*)
	Output_Params[1]:=MaxJointVel;
	Output_Params[2]:=0;
	Output_Params[3]:=0;
	Output_Params[4]:=0;
	Output_Params[5]:=0;
	Output_Params[6]:=0;


	(* If Values have change, Reinitialise Outputs*)

	IF FirstScan=0 OR 
		Robot.Outputs.MotionCommand.MoveSubIndex001 <> Output_Params[1] OR 
		Robot.Outputs.MotionCommand.MoveSubIndex002 <> Output_Params[2] OR 
		Robot.Outputs.MotionCommand.MoveSubIndex003 <> Output_Params[3] OR
		Robot.Outputs.MotionCommand.MoveSubIndex004 <> Output_Params[4] OR 
		Robot.Outputs.MotionCommand.MoveSubIndex005 <> Output_Params[5] OR 
		Robot.Outputs.MotionCommand.MoveSubIndex006 <> Output_Params[6] 
	THEN
		Buffered := FALSE;
		Sent := FALSE;
	END_IF;


	(*if not in legacy mode, Act Setpoint*)
	IF Robot.Outputs.MotionControl.MoveID <> 0 THEN
	    Robot.Outputs.MotionControl.SetPoint := TRUE;
	END_IF;

	(* To send _Move, send _Move ID *)
	IF NOT Buffered AND NOT Sent THEN
	    
	    Robot.Outputs.MotionCommand.MoveCommand	:= EnumToNum(Meca500Cmd#SetJointVelLimit);
	    Robot.Outputs.MotionCommand.MoveSubIndex001 := Output_Params[1];
		Robot.Outputs.MotionCommand.MoveSubIndex002 := Output_Params[2];
		Robot.Outputs.MotionCommand.MoveSubIndex003 := Output_Params[3];
		Robot.Outputs.MotionCommand.MoveSubIndex004 := Output_Params[4];
		Robot.Outputs.MotionCommand.MoveSubIndex005 := Output_Params[5];
		Robot.Outputs.MotionCommand.MoveSubIndex006 := Output_Params[6];
	    
	    IF ExternalStateControl THEN
	        IF ExternalMoveID <> 0 AND ExternalMoveID <> 33320 AND ExternalMoveID <> 33321 THEN
	            Robot.Outputs.MotionControl.MoveID := ExternalMoveID;
	            Sent := TRUE;
	        END_IF;
	        
	    ELSE (*Not External Control*)
	        IF Robot.Outputs.MotionControl.MoveID = 33320 THEN
	            Robot.Outputs.MotionControl.MoveID := 33321;
	        ELSIF Robot.Outputs.MotionControl.MoveID = 33321 THEN
	            Robot.Outputs.MotionControl.MoveID := 33320;
	        ELSIF Robot.Outputs.MotionControl.MoveID <> 33320 OR Robot.Outputs.MotionControl.MoveID <> 33321 THEN
	            Robot.Outputs.MotionControl.MoveID := 33320;
	        END_IF;
	        Sent := TRUE;
	    END_IF;
	END_IF;

	(* Check if command has been sent, if so, check if it was received *)
	IF Sent AND
	    Robot.Outputs.MotionCommand.MoveCommand = EnumToNum(Meca500Cmd#SetJointVelLimit) AND
	    Robot.Outputs.MotionCommand.MoveSubIndex001 = Output_Params[1] AND 
		Robot.Outputs.MotionCommand.MoveSubIndex002 = Output_Params[2] AND 
		Robot.Outputs.MotionCommand.MoveSubIndex003 = Output_Params[3] AND 
		Robot.Outputs.MotionCommand.MoveSubIndex004 = Output_Params[4] AND 
		Robot.Outputs.MotionCommand.MoveSubIndex005 = Output_Params[5] AND 
		Robot.Outputs.MotionCommand.MoveSubIndex006 = Output_Params[6] AND
		Robot.Inputs.Motion.MoveID = Robot.Outputs.MotionControl.MoveID 
	THEN
		 Buffered := TRUE;
	END_IF;


	(*If External _Move ID is equal to Internal, raise an error*)
	IF ExternalMoveID = 33320 OR ExternalMoveID = 33321 THEN
	    Error := TRUE;
	END_IF;

	FirstScan := TRUE;
ELSE
	FirstScan := False;
	Sent := FALSE;
	Buffered := FALSE;
END_IF;
END_FUNCTION_BLOCK

FUNCTION_BLOCK CalculateWRF
VAR
    x1 : REAL;
    x2 : REAL;
    x3 : REAL;
    y1 : REAL;
    y2 : REAL;
    y3 : REAL;
    z1 : REAL;
    z2 : REAL;
    z3 : REAL;
    ux : ARRAY[0..2] OF real;
    norm_ux : LREAL;
    uvx : ARRAY[0..2] OF Lreal;
    uy : ARRAY[0..2] OF lreal;
    norm_uy : LREAL;
    uvy : ARRAY[0..2] OF lreal;
    v13 : ARRAY[0..2] OF Lreal;
    norm_v13 : LREAL;
    uv13 : ARRAY[0..2] OF lreal;
    uz : ARRAY[0..2] OF Lreal;
    norm_uz : LREAL;
    uvz : ARRAY[0..2] OF lreal;
    beta : lreal;
    beta_deg : lreal;
    gamma : lreal;
    gamma_deg : lreal;
    alpha : lreal;
    alpha_deg : lreal;
END_VAR
VAR_INPUT
    Enable : BOOL;
    Point1 : ARRAY[0..2] OF real;
    Point2 : ARRAY[0..2] OF real;
    Point3 : ARRAY[0..2] OF real;
END_VAR
VAR_OUTPUT
    CalculatedWRF : ARRAY[0..5] OF lreal;
    Message : STRING[256];
END_VAR
//	Following the method available on Mecademic website : 
//	https://support.mecademic.com/en/support/solutions/articles/64000248048-how-do-i-calculate-the-wrf-using-a-3-point-method-

x1:=Point1[0];
x2:=Point2[0];
x3:=Point3[0];

y1:=Point1[1];
y2:=Point2[1];
y3:=Point3[1];

z1:=Point1[2];
z2:=Point2[2];
z3:=Point3[2];


ux[0]	:= x2 - x1;
ux[1]	:= y2 - y1;
ux[2]	:=	z2 - z1;
norm_ux := sqrt(EXPT(ux[0],2) + EXPT(ux[1],2) + EXPT(ux[2],2));

if norm_ux < 10 THEN
     Message:= ('Invalid Data: Points P2 and P1 are too close to each other');
else
     uvx[0] := ux[0]/norm_ux;
	 uvx[1] := ux[1]/norm_ux;
	 uvx[2] := ux[2]/norm_ux;
end_if;

v13[0] := x3 - x1;
v13[1] := y3 - y1;
v13[2] := z3 - z1;
norm_v13 := sqrt(EXPT(v13[0],2) + EXPT(v13[1],2) + EXPT(v13[2],2));

if norm_v13 < 10 THEN
    Message:= 'Invalid Data: Points P3 and P1 are too close to each other';
else 
     uv13[0] := v13[0]/norm_v13;
	 uv13[1] := v13[1]/norm_v13;
	 uv13[2] := v13[2]/norm_v13;
END_IF;

// uz = CrossProduct(uvx,uv13)
uz[0] := (uvx[1]*uv13[2])-(uvx[2]*uv13[1]);
uz[1] := (uvx[2]*uv13[0])-(uvx[0]*uv13[2]);
uz[2] := (uvx[0]*uv13[1])-(uvx[1]*uv13[0]);

// # the norm of this vector will be sin(theta), where theta is the angle between the two vectors, using the right-hand rule.
if NOT(norm_ux<10) and NOT (norm_v13 <10) THEN
     norm_uz := sqrt( EXPT(uz[0],2) + EXPT(uz[1],2) + EXPT(uz[2],2));
     uvz[0] := uz[0] / norm_uz;
	 uvz[1] := uz[1] / norm_uz;
	 uvz[2] := uz[2] / norm_uz;
END_IF;

// uvy = CrossProduct(uvz,uvx) 
uvy[0] := (uvz[1]*uvx[2])-(uvz[2]*uvx[1]);
uvy[1] := (uvz[2]*uvx[0])-(uvz[0]*uvx[2]);
uvy[2] := (uvz[0]*uvx[1])-(uvz[1]*uvx[0]) ;

// R = [ uvx,  uvy, uvz], where uvx, uvy and uvz are column vectors
if abs(uvz[0]) = 1 THEN
        beta_deg := uvz[0]*90;
        gamma := atan2(uvy[0],uvx[0]);
        gamma_deg := radtodeg(gamma);
        alpha_deg := 0;
else
        beta := asin(uvz[0]);
        beta_deg := radtodeg(beta);
        gamma := atan2(-uvy[0],uvx[0]);
        gamma_deg := radtodeg(gamma);
        alpha := atan2(-uvz[1],uvz[2]);
        alpha_deg := radtodeg(alpha) ;
END_IF;

CalculatedWRF[0] := x1;
CalculatedWRF[1] := y1;
CalculatedWRF[2] := z1;
CalculatedWRF[3] := alpha_deg;
CalculatedWRF[4] := beta_deg;
CalculatedWRF[5] := gamma_deg;
END_FUNCTION_BLOCK